
// ===== library: MasterCopy "ALARM_Simulation" =====

// folder: Rozdzial_8/Przyklad_8.3.1.1

FUNCTION_BLOCK "ALARM_Simulation"   // FB12, SCL
{ S7_Optimized_Access := 'TRUE' }
VERSION : 0.1
   VAR_INPUT
      Triggers : Array[1..10] of Bool;
      AlarmsDefinition : Array[1..10] of "alarmElement";
   END_VAR
   VAR_OUTPUT
      AlarmsStatus : Array[1..10] of "alarmStatus";
   END_VAR
   VAR_IN_OUT
      Acknowledge : Array[1..10] of Bool;
   END_VAR
   VAR
      AlarmsTexts : Array[1..10] of String;
      oldAck : Array[1..10] of Bool;
   END_VAR
   VAR_TEMP
      i : USInt;
      edge : Bool;
   END_VAR
BEGIN
   // Symulacja alarmów w sterowniku
   // W aktualnej wersji aplikacji SocialNotifier, alarmy definiowane są w bloku DB
   // i publikowane na serwerze w formie obiektów
   FOR #i := 1 TO 10 DO

       #edge := #Acknowledge[#i] AND NOT #oldAck[#i];
       #oldAck[#i] := #Acknowledge[#i];

       IF #Triggers[#i] THEN
           #AlarmsStatus[#i].type := #AlarmsDefinition[#i].type;
           #AlarmsStatus[#i].pendingAlarm := TRUE;
           #AlarmsStatus[#i].alarmText := CONCAT(IN1:=#AlarmsDefinition[#i].text, IN2:=#AlarmsDefinition[#i].parameter);
           IF #AlarmsDefinition[#i].mustBeAcknowledged THEN
               #AlarmsStatus[#i].ackRequired := TRUE;
           END_IF;
       ELSIF #Triggers[#i] = FALSE THEN
           IF #AlarmsDefinition[#i].mustBeAcknowledged THEN
               #AlarmsStatus[#i].pendingAlarm := FALSE;
               IF #edge THEN
                   #AlarmsStatus[#i].ackRequired := FALSE;
                   #AlarmsStatus[#i].alarmText := '';
                   #Acknowledge[#i] := FALSE;
                   #oldAck[#i] := #Acknowledge[#i];
               END_IF;

           ELSE
               #AlarmsStatus[#i].type := #AlarmsDefinition[#i].type;
               #AlarmsStatus[#i].pendingAlarm := FALSE;
               #AlarmsStatus[#i].ackRequired := FALSE;
               #AlarmsStatus[#i].alarmText := '';
           END_IF;

       END_IF;

   END_FOR;
END_FUNCTION_BLOCK

// ===== library: MasterCopy "ALARM_Control" =====

// folder: Rozdzial_8/Przyklad_8.3.1.1

DATA_BLOCK "ALARM_Control"   // DB24
{ S7_Optimized_Access := 'TRUE' }
VERSION : 0.1
   VAR
      AlarmTriggers : Array[1..10] of Bool;
      AlarmAck : Array[1..10] of Bool;
      AlarmsDefinition : Array[1..10] of "alarmElement";
      AlarmsStatus : Array[1..10] of "alarmStatus";
   END_VAR
BEGIN
   AlarmsDefinition[1].mustBeAcknowledged := true;
   AlarmsDefinition[1].text := 'Przekroczono dopuszczalny poziom cisnienia w zbiorniku. Aktualny poziom: ';
   AlarmsDefinition[2].mustBeAcknowledged := true;
   AlarmsDefinition[2].text := 'Przekroczono dopuszczalna temperature cieczy w zbiorniku. Aktualna wartosc: ';
   AlarmsDefinition[3].text := 'Blokada materialu w maszynie';
   AlarmsDefinition[4]."type" := 1;
   AlarmsDefinition[4].text := 'Wyzwolona funkcja ESTOP w maszynie';
   AlarmsDefinition[5]."type" := 2;
   AlarmsDefinition[5].text := 'Koniec zmiany - zatrzymano produkcje.';
END_DATA_BLOCK

// ===== library: MasterCopy "alarmElement" =====

// folder: Przyklad_8.3.1.1

TYPE "alarmElement"
   STRUCT
      "type" : USInt;   // 0=Alarm, 1=Ostrzezenie, 2=Informacja
      mustBeAcknowledged : Bool;   // TRUE=Wymaga potwierdzenia, FALSE=Nie wymaga potwierdzenia
      text : String;
      parameter : String;   // Dodatkowa wartosc dopisywana do alarmu
   END_STRUCT;
END_TYPE

// ===== library: MasterCopy "alarmStatus" =====

// folder: Przyklad_8.3.1.1

TYPE "alarmStatus"
   STRUCT
      "type" : USInt;   // 0=Alarm, 1=Ostrzezenie, 2=Informacja
      pendingAlarm : Bool;
      ackRequired : Bool;
      alarmText : String;
   END_STRUCT;
END_TYPE